FUNCTION_BLOCK FB_LightToggleCommand IMPLEMENTS I_Command
VAR_INPUT
END_VAR
VAR_OUTPUT
END_VAR
VAR
	// Reference to the Light that should be switched on.
	iLight: I_Switchable;
	bState: BOOL;
END_VAR

METHOD Execute
IF (iLight <> 0) THEN
	IF (iLight.Active) THEN
		THIS^.iLight.Off();
	ELSE
		THIS^.iLight.On();
	END_IF
END_IF
END_METHOD

METHOD FB_init : BOOL
VAR_INPUT
	bInitRetains : BOOL; // if TRUE, the retain variables are initialized (warm start / cold start)
	bInCopyCode : BOOL;  // if TRUE, the instance afterwards gets moved into the copy code (online change)
	iSwitchable : I_Switchable;
END_VAR
IF (iSwitchable <> 0) THEN
	THIS^.iLight := iSwitchable;
END_IF
END_METHOD

END_FUNCTION_BLOCK

(* stored: Version 1.1.0.1, ProductVersion 3.1.4024.5
   POU FB_LightToggleCommand: Id {1be5fb85-af3c-4300-8483-79076bf1e423}, SpecialFunc None
   Method Execute: Id {c547f585-8956-4230-aac2-8ae79a234e86}
   Method FB_init: Id {a88efd9c-4de7-4cff-9b85-8987f64460cc} *)
